PROGRAM _01_MAIN
(****************************************************************************)
//GENERAL PROGRAMM
//	- Call Sub-Programs
//
//	04.09.2019/Dj
//
//	Version:
(****************************************************************************)
VAR
END_VAR

//--------------------------------------------------------------------------
// PROGRAM CALLS
//--------------------------------------------------------------------------
//Allgemein
//_02_SAFETY();
//_05_FLAGS( xIN_AIR:=FALSE, xIN_btRES_TEMP:=HMI.btArMain[8]);

//HMI
//_10_HMI();

//AUTO
//_20_AUTO(xIN_Quit:= _14_STATE._FB_btQUIT.pbtIN^.rtrig , enIN_State:= );

END_PROGRAM

(* stored: Version 1.1.0.1, ProductVersion 3.1.4024.6
   POU _01_MAIN: Id {f3967eba-7efc-4619-8471-a18348d0943c}, SpecialFunc None *)
